{attribute addProperty BoxType "EL6002-0000-0019"}
{attribute addProperty Id "COM_TxPDO_Map_Inputs_ChannelAT %I*ARRAY[0..23] OF COM_TxPDO_Map_Inputs_Channel_85D1D733384480COM_RxPDO_Map_Outputs_ChannelAT %Q*ARRAY[0..23] OF COM_RxPDO_Map_Outputs_Channel_85BCA431384480WcStateAT %I*WcState_98A4DF7520.250InfoDataAT %I*InfoData_BC63D37F80100"}
{attribute addProperty CRC "3311090797"}
{attribute addProperty SizeInBites "850"}
{attribute addProperty SizeInBytes "106.25"}
TYPE EL6002_CC591D2E :
STRUCT
	{attribute addProperty Name "COM_TxPDO_Map_Inputs_Channel"}
	COM_TxPDO_Map_Inputs_Channel : ARRAY[0..23] OF COM_TxPDO_Map_Inputs_Channel_85D1D733;
	{attribute addProperty Name "COM_RxPDO_Map_Outputs_Channel"}
	COM_RxPDO_Map_Outputs_Channel : ARRAY[0..23] OF COM_RxPDO_Map_Outputs_Channel_85BCA431;
	{attribute addProperty Name "WcState"}
	WcState : WcState_98A4DF75;
	{attribute addProperty Name "InfoData"}
	InfoData : InfoData_BC63D37F;
END_STRUCT
END_TYPE

(* stored: Version 1.2.0.0, ProductVersion 3.1.4024.9
   DUT EL6002_CC591D2E: Id {9ae9dfb2-9081-0b67-3a9e-b63bd89796c6} *)
